// TIA Portal V18 export
TYPE "typePositions"
// stored: IsFailsafeCompliant false
   STRUCT
      M1Z : Real;
      M2Y : Real;
      M3X : Real;
      M4O1 : Real;
      M5O2 : Real;
   END_STRUCT;
END_TYPE
